FUNCTION_BLOCK ABSTRACT CUBaseSuspend EXTENDS TcoTaskedSequencer
VAR
	_done:BOOL;

END_VAR

PROPERTY Done : bool
GET
Done := _done;
END_GET
END_PROPERTY

METHOD PUBLIC OnStart
_done:=FALSE;
END_METHOD

PROPERTY StationBase : REFERENCE TO CuBase
GET
VAR
    _station : POINTER TO CuBase;
END_VAR
IF __QUERYPOINTER(Parent, _station) THEN // Check if _Parent is Station001
    StationBase REF= _station^;              // If the check is successful dereference a pointer. simlar to THIS^ or SUPER^
END_IF
END_GET
END_PROPERTY

END_FUNCTION_BLOCK

(* stored: Version 1.1.0.1
   POU CUBaseSuspend: Id {186121a4-6f79-4bd8-9c72-9cb4d29ea7ca}, SpecialFunc None
   Property Done: Id {5a22d587-5150-4d6f-a4dd-4eb67fd1aa1b}
   Get Get: Id {1450861f-0942-49e9-a6a4-490ac06bb997}
   Method OnStart: Id {b57d8d71-ae82-45fe-9fe9-f07ca10c4c78}
   Property StationBase: Id {b74542a3-cffc-49be-bea0-b126e11ecbb7}
   Get Get: Id {9e31189c-64d9-4e24-84e1-c3db17654050} *)
